{attribute 'qualified_only'}
VAR_GLOBAL
	lrRawTemp AT %I*			: INT;
	lrHotendTemp 				: LREAL;
	iHotendPowerLevel AT %Q*	: INT;
	bEnableHotend AT %Q*		: BOOL;
	bFan AT %Q*					: BOOL;
	bExcuteButton AT %I*		: BOOL;
END_VAR

(* stored: Version 1.1.0.1, ProductVersion 3.1.4024.2
   GVL GVL_IO: Id {2dc9d395-068a-4ece-b874-33348ddfb31a} *)
